//{warning 'CONVERSION MESSAGE: This text contained unprintable characters, that have been deleted'.}
TYPE ST_HMI_CylinderCtrl :
STRUCT
	stDisable			: ST_HMI_Buttons;
	stRelease			: ST_HMI_Buttons;
	eCommand			: E_CYLINDER_Position;

END_STRUCT
END_TYPE

(* stored: Version 1.1.0.1
   DUT ST_HMI_CylinderCtrl: Id {000c6fef-d352-402d-b32f-174268bed49d} *)
